// TwinCAT 3 PLC project test
// ProgramVersion: 3.1.4024.0
// libraries:
//   Tc2_Standard, * (Beckhoff Automation GmbH)
//   Tc2_System, * (Beckhoff Automation GmbH)
//   Tc3_Module, * (Beckhoff Automation GmbH)
// project tree:
//   / PlcTask.TcTTO
//   POUs/ MAIN.TcPOU
// real-time tasks:
//   TASK PlcTask: cycle T#10ms, priority 20, ADS port 350
// I/O:
//   DEVICE Device 2 (EtherCAT), AmsNetId 10.1.42.124.3.1
//     Box 1 (NETX 90-RE/ECS) [NETX 90-RE/ECS]
// variable links:
//   test/test Instance <-> Device 2 (EtherCAT)/Box 1 (NETX 90-RE/ECS)
//     PlcTask Inputs/MAIN.uiTxByte0 <-> TxPDO 1A00/1 Byte In (0)
//     PlcTask Inputs/MAIN.uiTxByte1 <-> TxPDO 1A00/1 Byte In (1)
//     PlcTask Inputs/MAIN.uiTxByte2 <-> TxPDO 1A00/1 Byte In (2)
//     PlcTask Outputs/MAIN.uiTrigger <-> RxPDO 1600/1 Byte Out (5)

CONFIGURATION test
    RESOURCE PLC ON TwinCAT3
        TASK PlcTask(INTERVAL := T#10ms, PRIORITY := 20);
        PROGRAM MAIN WITH PlcTask : MAIN;
    END_RESOURCE
END_CONFIGURATION

// ---- POUs/MAIN.TcPOU
PROGRAM MAIN
VAR
    (*– I/O Mappings –*)
    uiTrigger      AT %QB5   : USINT;    // RxPDO 0x1600 Byte Out 5 trigger :contentReference[oaicite:0]{index=0}
    uiTxByte0      AT %IB0   : USINT;   // TxPDO byte 0 → process-image byte 0 :contentReference[oaicite:1]{index=1}
    uiTxByte1      AT %IB1   : USINT;   // TxPDO byte 1 → process-image byte 1 :contentReference[oaicite:2]{index=2}
    uiTxByte2      AT %IB2   : USINT;   // TxPDO byte 2 → process-image byte 2 :contentReference[oaicite:3]{index=3}

    (*– State & File I/O –*)
    prevTrig       : BOOL := FALSE;     // previous scan trigger state :contentReference[oaicite:4]{index=4}
    loggingActive  : BOOL := FALSE;     // TRUE between rising/falling edges :contentReference[oaicite:5]{index=5}

    fbOpen         : FB_FileOpen;       // opens or creates the CSV file :contentReference[oaicite:6]{index=6}
    fbWrite        : FB_FileWrite;      // writes data into the file :contentReference[oaicite:7]{index=7}
	fbRead         : FB_FileRead;
	fbclose        : FB_FileClose;

    hSrcFile          : UINT;              // handle returned by FB_FileOpen (UINT) :contentReference[oaicite:8]{index=8}
    ts             : ULINT;             // 100 ns-resolution timestamp :contentReference[oaicite:9]{index=9}
    sLine          : STRING(120);       // formatted CSV line buffer :contentReference[oaicite:10]{index=10}
    bytesWritten   : UDINT;             // number of bytes actually written
	
	bTrigger       : BOOL;
	nErrId: UDINT;
	bError: BOOL;
	Step: UDINT;
	openDone : BOOl :=FALSE;
	sLine_len: UDINT;
END_VAR


// === ONE-TIME INITIALIZATION ===
(* Open CSV file for append; MODE_WRITE|MODE_CREATE = 16#0002 *)  
IF NOT opendone THEN
	fbOpen(  
		sPathName := 'C:\Users\parnika.gupta\Documents\twincat_log.csv',
		nMode     := 16#000C, //FOPEN_MODEAPPEND OR FOPEN_MODEPLUS OR FOPEN_MODETEXT,
		bExecute := TRUE,
		tTimeout := T#1S,
	);
	openDone := TRUE;
END_IF

fbOpen.bExecute := FALSE;// reset execute flag per FB_FileOpen state machine :contentReference[oaicite:12]{index=12}  
IF NOT fbOpen.bBusy AND NOT openDone THEN 
   IF fbOpen.bError THEN 
		nErrId := fbOpen.nErrId; 
		bError := TRUE; 
		Step := 50; 
   ELSE 
		hSrcFile := fbOpen.hFile; // store the file handle for writes :contentReference[oaicite:11]{index=11}
		Step := Step + 1; 
   END_IF 
END_IF 
// On each cycle, evaluate uiTrigger:
//   • If uiTrigger ≠ 0 → bTriggerBool := TRUE
//   • If uiTrigger = 0 → bTriggerBool := FALSE
bTrigger := 1; //(uiTrigger <> 0);

// === CYCLIC TASK: EDGE DETECTION & LOGGING ===
(* 1) Rising edge: trigger from 0→1 → start logging *)  
IF bTrigger AND NOT prevTrig THEN  
    loggingActive := TRUE;  
END_IF  

(* 2) Falling edge: trigger from 1→0 → stop logging *)  
IF NOT bTrigger AND prevTrig THEN  
    loggingActive := FALSE;  
END_IF  

prevTrig := bTrigger;   // update previous trigger for next cycle :contentReference[oaicite:13]{index=13}  

// 3) While loggingActive, capture timestamp & write CSV  
IF openDone AND loggingActive THEN  
    ts := F_GetSystemTime();  // read 64-bit OS time (100 ns units) :contentReference[oaicite:14]{index=14}  

    // build comma-separated line: "<ts>,<b0>,<b1>,<b2>\r\n"  
    sLine := CONCAT(
            CONCAT(
              CONCAT(
                CONCAT(
                  CONCAT( TO_STRING(ts), ',' ),  // ts → STRING
                  TO_STRING(uiTxByte0)           // byte0 → STRING
                ),
                ','                              // literal separator
              ),
              TO_STRING(uiTxByte1)               // byte1 → STRING
            ),
            CONCAT(
              CONCAT( ',', TO_STRING(uiTxByte2) ),  // ',', byte2
              '\r\n'                                // newline
            ));
		// :contentReference[oaicite:15]{index=15}  

    // append the line to the file  	
	sLine_len := INT_TO_UDINT(LEN(sLine));
	IF sLine_len >4 THEN
		fbWrite(  
			hFile       := hSrcFile, // file handle (UINT) :contentReference[oaicite:16]{index=16}  
			pWriteBuff  := ADR(sLine),          // pointer to data buffer :contentReference[oaicite:17]{index=17}  
			cbWriteLen  := sLine_len,          // number of chars to write :contentReference[oaicite:18]{index=18}  
			bExecute    := TRUE,                // trigger write on edge :contentReference[oaicite:19]{index=19}
			tTimeout := T#1S,
		);  
		fbWrite.bExecute := FALSE;          // reset for next write :contentReference[oaicite:20]{index=20}  
		//fbWrite( bExecute := FALSE ); 
		(*IF openDone AND (hSrcFile <> 0) AND NOT fbWrite.bBusy THEN 
		   IF fbWrite.bError THEN 
				nErrId := fbWrite.nErrId; 
				bError := TRUE; 
				Step := 50; 
		   ELSE 
				IF fbRead.bEOF THEN (* Check if the EOF flag ist set *) 
					 Step := 50;     (* Cleanup: close the destination and source files *) 
				ELSE 
					 Step := 5; (* Repeat reading/writing *) 
				END_IF
			END_IF
		END_IF*)
	END_IF

	
END_IF  


fbClose(
	hFile := hSrcFile,
	bExecute := TRUE,
	tTimeout := T#1S,
);

END_PROGRAM
